(* IEC 61131-3 sources: volt/packages/volt-lsp-iec/test-corpus/bakon-nano/Device/Plc Logic/Application/POUs/MachineControl (part 2) *)

(* ---- MACH_MCL_ModeControl.pou ---- *)
PROGRAM MACH_MCL_ModeControl
VAR
	(* Temporary Variables *)
	bPulseStepCounter	: BOOL;
	bRecipeLoaded		: BOOL;
	tDisableDrives		: TON;
	tonStartButton		: TON;
END_VAR
%LANGUAGE ST
(*************************************************************************
 *
 * Application name				: Snijmachine
 * Module name					: MACH_MCL_ModeControl
 * Version number module		: 0.30
 *
 *
 *						Copyright (c) Bakon 2009
 *						Goes, The Netherlands
 *
 *
 * All rights are reserved. Reproduction in whole or in part is prohibited
 * without the written consent of the copyright owner.
 *
 *************************************************************************)

(*****************************************************************************
 * HISTORY
 *****************************************************************************
 * Update		: 0.20
 * Author		: K.Kole (KOOLE CONTROLS)
 * Changes	: 0.10:	Force to state WaitForInit changed
 *						Condition "bEnableMachine" added in state "WaitForConditioning"
 *				  0.20:	Blockingcounter implemented
 *				  0.30:  Ondelay added for bit g_HMI_bRecipeLoaded in order to avoid
 *						a error in state Wait_For_Automatic
 *****************************************************************************)

	(****************************************************************)
	(*  Mode Control is the central control part of the machines.	*)
	(*  It receives and sends signals from and to the HMI and		 *)
	(*  Handles the signals to and from the machine					  *)
	(****************************************************************)

	(* Hold automatic when ErrorCategory3 *)
	IF			g_sMACH.ERH.bErrorCategory3
	THEN
				g_sMACH.MCL.bHoldOnErrorCat3 := TRUE;
	END_IF
	IF	  	NOT g_sMACH.ERH.bErrorCategory3
		AND	g_HMI_MachCommand.CMD.bStartCycle
	THEN
				 g_sMACH.MCL.bHoldOnErrorCat3 := FALSE;
	END_IF

	(* Stop at end of cycle when ErrorCategory2 *)
	IF				g_sMACH.ERH.bErrorCategory2
	THEN
					g_sMACH.MCL.bStopOnErrorCat2 := TRUE;
	END_IF
	IF	  	NOT	g_sMACH.ERH.bErrorCategory2
		AND NOT	g_sMACH.MCL.bActAutomatic
	THEN
					g_sMACH.MCL.bStopOnErrorCat2 := FALSE;
	END_IF

	(* Stop at end of cycle *)
	IF 	g_HMI_MachCommand.CMD.bStopCycle
	THEN
		g_sMACH.MCL.bStopEndOfCycle := TRUE;
	END_IF
	IF NOT g_sMACH.MCL.bActAutomatic
	THEN
		g_sMACH.MCL.bStopEndOfCycle := FALSE;
	END_IF

	bRecipeLoaded := (g_HMI_sRecipeName <> 'new recipe') AND (g_HMI_sRecipeName <> '');

	(* Recipe downloaded. *)
(*	IF			bRecipeLoaded
		AND (	MACH.MCL.bStateMainSwitchedOn
			OR MACH.MCL.bStateWaitForInit
			OR MACH.MCL.bStateInit
			OR MACH.MCL.bStateWaitForRecipe)
	THEN
		MACH.MCL.bRecipeExecuted := TRUE;
	END_IF
*)
	(* Force StateWaitForAutomatic *)
	IF		  		g_bFirstCycle
		OR NOT 	g_bDI_ES_DirectOK
		OR		g_sMACH.ERR.bTableMovementNotAllowed		// Severe error, chance of damaging the knife
		OR		g_sMACH.ERR.bRAxisMovementNotAllowed		// Severe error, chance of damaging the knife
		OR		g_sMACH.ERR.bZAxisMovementNotAllowed		// Severe error, chance of damaging the knife
		OR		(g_sMACH.ERH.bErrorCategory4
		AND NOT	g_sMACH.MCL.bActManual
		//AND (NOT g_sMACH.MCL.bActAutomatic OR g_bSUB_CleanKnifeStart)
		AND		g_sMACH.MCL.nStepCounter <> StateWaitForAutomatic)
	THEN
				 g_sMACH.MCL.nStepCounter := StateWaitForAutomatic;
	//ELSIF		g_sMACH.ERH.bErrorCategory4			(* Force StateWaitForAuto *)
	//	AND 	g_sMACH.MCL.bActAutomatic
	//	AND NOT	g_bSUB_CleanKnifeStart
	//THEN
	//			 g_sMACH.MCL.nStepCounter := StateWaitForAutomatic;
	END_IF

	(* detect change of state *)
	bPulseStepCounter				:= g_sMACH.MCL.nStepCounter <> g_sMACH.MCL.nOldStepCounter;
	g_sMACH.MCL.nOldStepCounter	:= g_sMACH.MCL.nStepCounter;

IF bPulseStepCounter THEN
	{warning 'Disabled for compatibility SVE'}
	//g_Logger.Write(0, CONCAT('Modecontrol changed to state ', INT_TO_STRING(g_sMACH.MCL.nStepCounter)), 'MACH_MCL_ModeControl');
END_IF

tonStartButton(IN:= g_bDI_StartButton, PT:= T#500MS, Q=> , ET=> );

CASE g_sMACH.MCL.nStepCounter OF
	(* ------------------------------------------------------------------------------
	 * S000 StateMainSwitchedOn
	 *		Reset all Mode Control variables
	 * ------------------------------------------------------------------------------ *)
	StateMainSwitchedOn:

		(* On Entry *)
		IF bPulseStepCounter
		THEN
			g_sMACH.MCL.bActInitialise				:= FALSE;
			g_sMACH.MCL.bActConditioning			:= FALSE;
			g_sMACH.MCL.bActAutomatic			:= FALSE;
			g_sMACH.MCL.bActManual				:= FALSE;
			g_sMACH.MCL.bActCleaning				:= FALSE;
			g_sMACH.MCL.bHoldOnRequest		:= FALSE;
			g_sMACH.MCL.bStopEndOfCycle		:= FALSE;

			(*g_sMACH.MCL.bInitExecuted				:= FALSE; *)
			g_sMACH.MCL.bRecipeExecuted		:= FALSE;
			g_HMI_MachCommand.CMD.bStartManual					:= FALSE;
			g_HMI_MachCommand.CMD.bStartCleaning				:= FALSE;
		  	g_HMI_MachCommand.CMD.bStartCycle				:= FALSE;
		END_IF

		(* Continous actions *)

		(* Transitions *)
		IF				g_bDI_ES_DirectOK
			AND NOT	g_sMACH.ERH.bErrorCategory4
		THEN
			g_sMACH.MCL.nStepCounter := StateWaitForAutomatic;(* StateWaitForInit; *)
			(* On Exit *)
		ELSIF			g_bDI_ES_DirectOK
			AND		g_HMI_MachCommand.CMD.bStartManual
		THEN
			g_sMACH.MCL.nStepCounter := StateManual;
		END_IF

	(* ------------------------------------------------------------------------------
	 * S001 StateWaitForInit
	 *		Wait for init button (No error present )
	 * ------------------------------------------------------------------------------ *)
	StateWaitForInit:

		(* On Entry *)
		IF bPulseStepCounter
		THEN
			(*g_sMACH.MCL.bInitExecuted		:= FALSE; *)
			g_sMACH.MCL.bActInitialise		:= FALSE;
			g_sMACH.MCL.bActConditioning := FALSE;
			g_sMACH.MCL.bActAutomatic	:= FALSE;
			g_sMACH.MCL.bActManual		:= FALSE;
			g_sMACH.MCL.bActCleaning		:= FALSE;
			g_HMI_MachCommand.CMD.bStartManual			:= FALSE;
			g_HMI_MachCommand.CMD.bStartCleaning		:= FALSE;
			g_HMI_MachCommand.CMD.bStartCycle		:= FALSE;

			g_sMACH.MCL.bHoldOnRequest		:= FALSE;
			g_sMACH.MCL.bStopEndOfCycle		:= FALSE;

			tDisableDrives(IN:=FALSE);
			(*g_sMACH.MCL.bRecipeExecuted		:= FALSE; Storing weggelaten dd 1 juni 2011 *)
		END_IF

		(* Continous actions *)
		tDisableDrives(IN:=TRUE, PT:= t#1500ms);
		IF tDisableDrives.Q THEN								(* In AUT, MAN, INI cycles g_uControl_xxx.bAutomatic etc. is reset *)
			g_uControl_X_Axis.bEnableDrive	:= FALSE;			(* Resetting the bEnableDrive bit must be delayed *)
			g_uControl_Y_Axis.bEnableDrive	:= FALSE;
			{warning 'SVE - Check this change}
			//g_uControl_Front_Axis.bEnableDrive	:= g_uStatus_Front_Axis.nStateAxis = 3 OR g_uStatus_Front_Axis.nStateAxis <= 1;			(* Resetting the bEnableDrive bit must be delayed *)
			//g_uControl_Rear_Axis.bEnableDrive	:= g_uStatus_Rear_Axis.nStateAxis = 3 OR g_uStatus_Rear_Axis.nStateAxis <= 1;
			g_uControl_Front_Axis.bEnableDrive := g_uStatus_Front_Axis.eStateAxis <= L_MC1P_AXIS_STATE.StandStill;		//Standstill, Disabled or Errorstop
			g_uControl_Rear_Axis.bEnableDrive := g_uStatus_Rear_Axis.eStateAxis <= L_MC1P_AXIS_STATE.StandStill;		//Standstill, Disabled or Errorstop
			g_uControl_Z_Axis.bEnableDrive	:= FALSE;
			g_uControl_R_Axis.bEnableDrive	:= FALSE;
		END_IF
		(*g_sMACH.ERR.bMoldWarningMold := (NOT FUN_CHECK_MOLD(g_bDI_MoldLeftPresent, g_bDI_MoldRightPresent,(g_HMI_RCP_Parameters.nProductType = Prod_Round),
																			g_bDI_MoldDetection1_1, g_bDI_MoldDetection1_2, g_bDI_MoldDetection1_3,
																			g_bDI_MoldDetection2_1, g_bDI_MoldDetection2_2, g_bDI_MoldDetection2_3,
																			g_HMI_RCP_Parameters.nMaxMoldParts) ) AND (bRecipeLoaded); *)

		(* Transitions *)
		IF 	NOT		g_sMACH.ERH.bError234Active
			AND NOT g_uStatus_X_Axis.bDriveEnabled
			AND NOT g_uStatus_Y_Axis.bDriveEnabled
			AND NOT g_uStatus_Front_Axis.bDriveEnabled
			AND NOT g_uStatus_Rear_Axis.bDriveEnabled
			AND NOT g_uStatus_Z_Axis.bDriveEnabled
			AND NOT g_uStatus_R_Axis.bDriveEnabled
			AND	g_uStatus_R_Axis.bHomePositionAvailable
			AND	(g_HMI_MachCommand.CMD.bStartCycle OR (tonStartButton.Q AND g_HMI_MachCommand.bScanMode))
		THEN
			g_sMACH.MCL.nStepCounter := StateInit;
			(* On Exit *)
		ELSIF g_HMI_MachCommand.CMD.bStartManual						(* Manual *)
		THEN
			g_sMACH.MCL.nStepCounter := StateManual;
		END_IF

	(* ------------------------------------------------------------------------------
	 * S002 StateInit
	 *		Initialising busy
	 * ------------------------------------------------------------------------------ *)
	StateInit:

		(* On Entry *)
		IF bPulseStepCounter
		THEN
			;(*g_sMACH.MCL.bInitExecuted := FALSE; *)
		END_IF

		(* Continous actions *)
		g_sMACH.MCL.bActInitialise := TRUE;

		(* Transitions *)
		IF g_sMACH.uINI.bInitialiseReady
		THEN
			g_sMACH.MCL.nStepCounter := StateWaitForRecipe;
			(* On Exit *)
			g_sMACH.MCL.bActInitialise := FALSE;
			(*g_sMACH.MCL.bInitExecuted  := TRUE; *)
		END_IF

	(* ------------------------------------------------------------------------------
	 * S003 StateWaitForRecipe
	 *		Wait for recipe download
	 * ------------------------------------------------------------------------------ *)
	StateWaitForRecipe:

		(* On Entry *)

		(* Continous actions *)

		(* Transitions *)
		IF bRecipeLoaded						(* Recipe loaded *)
		THEN
			g_sMACH.MCL.nStepCounter := StateWaitForAutomatic;
		ELSIF g_HMI_MachCommand.CMD.bStartManual						(* Manual *)
		THEN
			g_sMACH.MCL.nStepCounter := StateManual;
		ELSIF g_HMI_MachCommand.CMD.bStartCleaning					(* Cleaning *)
		THEN
			g_sMACH.MCL.nStepCounter := StateCleaning;
		END_IF

	(* ------------------------------------------------------------------------------
	 * S004 StateWaitForConditioning
	 *		Wait for start button
	 * ------------------------------------------------------------------------------ *)
(*	StateWaitForConditioning:

		(* On Entry *)
		IF bPulseStepCounter
		THEN
			g_sMACH.MCL.bConditioningExecuted := FALSE;
		END_IF

		(* Continous actions *)

		(* Transitions *)
		IF	g_HMI_MachCommand.CMD.bStartCycle THEN
			g_sMACH.MCL.nStepCounter := StateWaitForAutomatic;
		ELSIF g_HMI_MachCommand.CMD.bStartCycle				  (* Conditioning *)
		THEN
			g_sMACH.MCL.nStepCounter := StateConditioning;
		ELSIF g_sMACH.MCL.bStartInitialise		(* Initialise *)
		THEN
			g_sMACH.MCL.nStepCounter := StateInit;
		ELSIF g_sMACH.MCL.bStartManual			 (* Manual *)
		THEN
			g_sMACH.MCL.nStepCounter := StateManual;
		ELSIF g_sMACH.MCL.bStartCleaning						(* Cleaning *)
		THEN
			g_sMACH.MCL.nStepCounter := StateCleaning;
		END_IF

	(* ------------------------------------------------------------------------------
	 * S005 StateConditioning
	 *		Conditioning busy
	 * ------------------------------------------------------------------------------ *)
	StateConditioning:

		(* On Entry *)
		IF bPulseStepCounter
		THEN
			g_sMACH.MCL.bConditioningExecuted := FALSE;
		END_IF

		(* Continous actions *)
		g_sMACH.MCL.bActConditioning := TRUE;

		(* Transitions *)
		IF (*g_sMACH.CON.BCONDITIONINGREADY*) TRUE
		THEN
			g_sMACH.MCL.nStepCounter := StateWaitForAutomatic;
			(* On Exit *)
			g_sMACH.MCL.bActConditioning		:= FALSE;
			g_sMACH.MCL.bConditioningExecuted := TRUE;
		END_IF
*)
	(* ------------------------------------------------------------------------------
	 * S006 StateWaitForAutomatic
	 *		Wait for start button
	 * ------------------------------------------------------------------------------ *)
	StateWaitForAutomatic:

		(* On Entry *)
		IF bPulseStepCounter
		THEN
			g_sMACH.MCL.bActInitialise		:= FALSE;
			g_sMACH.MCL.bActConditioning := FALSE;
			g_sMACH.MCL.bActAutomatic	:= FALSE;
			g_sMACH.MCL.bActManual		:= FALSE;
			g_sMACH.MCL.bActCleaning		:= FALSE;
			g_HMI_MachCommand.CMD.bStartManual			:= FALSE;
			g_HMI_MachCommand.CMD.bStartCleaning		:= FALSE;
			g_HMI_MachCommand.CMD.bStartCycle		:= FALSE;

			g_sMACH.MCL.bHoldOnRequest		:= FALSE;
			g_sMACH.MCL.bStopEndOfCycle		:= FALSE;

			tDisableDrives(IN:=FALSE);
		END_IF

		(* Continous actions *)
		tDisableDrives(IN:=TRUE, PT:= t#1500ms);
		IF tDisableDrives.Q THEN									(* In AUT, MAN, INI cycles g_uControl_xxx.bAutomatic etc. is reset *)
			g_uControl_X_Axis.bEnableDrive	:= FALSE;			(* Resetting the bEnableDrive bit must be delayed *)
			g_uControl_Y_Axis.bEnableDrive	:= FALSE;
			{warning 'SVE - Check this change}
			//g_uControl_Front_Axis.bEnableDrive	:= g_uStatus_Front_Axis.nStateAxis <> 3 AND g_uStatus_Front_Axis.nStateAxis >= 2;			(* Resetting the bEnableDrive bit must be delayed *)
			//g_uControl_Rear_Axis.bEnableDrive	:= g_uStatus_Rear_Axis.nStateAxis <> 3 AND g_uStatus_Rear_Axis.nStateAxis >= 2;
			g_uControl_Front_Axis.bEnableDrive := g_uStatus_Front_Axis.eStateAxis > L_MC1P_AXIS_STATE.StandStill;	//XX_Motion
			g_uControl_Rear_Axis.bEnableDrive := g_uStatus_Rear_Axis.eStateAxis > L_MC1P_AXIS_STATE.StandStill;	//XX_Motion
			g_uControl_Z_Axis.bEnableDrive	:= FALSE;
			g_uControl_R_Axis.bEnableDrive	:= FALSE;
		END_IF;

		(* Transitions *)
		IF				(g_HMI_MachCommand.CMD.bStartCycle  OR (tonStartButton.Q AND g_HMI_MachCommand.bScanMode))					(* Start auto cycle *)
			AND NOT	g_sMACH.MCL.bStopOnErrorCat2
			AND NOT	g_sMACH.MCL.bHoldOnErrorCat3
			AND		g_bAxis_FrontSet								(* Axis referenced to zero (in manual page) *)
			AND		g_bAxis_RearSet								(* Axis referenced to zero (in manual page) *)
			AND		g_bAxis_RSet									(* Axis referenced to zero (in manual page) *)
			AND		((g_sHMI_CountersInfinite.dnHourCount <= g_HMI_MCH_dnBlockCounter) OR (g_HMI_MCH_dnBlockCounter = 0))
		THEN
			g_sMACH.MCL.nStepCounter := StateAutomatic;
		ELSIF g_HMI_MachCommand.CMD.bStartManual								(* Manual *)
		THEN
			g_sMACH.MCL.nStepCounter := StateManual;
		ELSIF g_HMI_MachCommand.CMD.bStartCleaning							(* Cleaning *)
		THEN
			g_sMACH.MCL.nStepCounter := StateCleaning;
		END_IF

	(* ------------------------------------------------------------------------------
	 * S007 StateAutomatic
	 *		Automatic busy
	 * ------------------------------------------------------------------------------ *)
	StateAutomatic:

		(* On Entry *)

		(* Continous actions *)
		g_sMACH.MCL.bActAutomatic := TRUE;
		IF	g_HMI_MachCommand.CMD.bPauseCycle
		THEN
			g_sMACH.MCL.bHoldOnRequest := TRUE;
		END_IF
		IF	g_HMI_MachCommand.CMD.bStartCycle
		THEN
			g_sMACH.MCL.bHoldOnRequest := FALSE;
		END_IF

		(* Transitions *)
		IF g_sMACH.AUT.bAutomaticReady
		THEN
			g_sMACH.MCL.nStepCounter := StateWaitForAutomatic;
			(* On Exit *)
			g_sMACH.MCL.bActAutomatic			:= FALSE;
			g_sMACH.MCL.bHoldOnRequest		:= FALSE;
		END_IF

	(* ------------------------------------------------------------------------------
	 * S008 StateManual
	 *		Manual mode busy
	 * ------------------------------------------------------------------------------ *)
	StateManual:

		(* On Entry *)
		IF bPulseStepCounter
		THEN
			g_sMACH.MCL.bActManual := TRUE;
		END_IF

		(* Continous actions *)
		g_HMI_MachCommand.CMD.bStartManual	:= FALSE;
		IF 	g_HMI_MachCommand.CMD.bStopManual
		THEN
			g_sMACH.MCL.bStopEndOfCycle := TRUE;
		END_IF

		(* Transitions *)
		IF g_sMACH.MAN.bManualReady
		THEN
			g_sMACH.MCL.bActManual := FALSE;
			g_sMACH.MCL.nStepCounter := StateWaitForAutomatic;	(* StateWaitForInit; *)
		END_IF

	(* ------------------------------------------------------------------------------
	 * S009 StateCleaning
	 *		Cleaning mode busy
	 * ------------------------------------------------------------------------------ *)
	StateCleaning:

		(* On Entry *)
		IF bPulseStepCounter
		THEN
			g_sMACH.MCL.bActCleaning := TRUE;
			g_HMI_MachCommand.CMD.bStopCleaning	:= FALSE;
		END_IF

		(* Continous actions *)
		IF	g_HMI_MachCommand.CMD.bStopCleaning
		THEN
			g_sMACH.MCL.bStopEndOfCycle := TRUE;
		END_IF

		(* Transitions *)
		IF	g_sMACH.CLN.bCleaningReady
		THEN
			g_sMACH.MCL.bActCleaning := FALSE;
			g_HMI_MachCommand.CMD.bStopCleaning	:= FALSE;
			g_sMACH.MCL.nStepCounter := StateWaitForAutomatic;	(*StateWaitForInit; *)
		END_IF

	END_CASE

END_PROGRAM

(* ---- MACH_MIS_Miscellaneous.pou ---- *)
PROGRAM MACH_MIS_Miscellaneous
VAR
	TONMinute: TON;
	bMinute	: BOOL;

END_VAR
%LANGUAGE ST
(* Machine producing hours *)
TONMinute(IN:=g_sMACH.AUT.bActAutomatic AND NOT bMinute, PT:=T#60s);
bMinute := TONMinute.Q;
IF bMinute THEN
	 g_sHMI_CountersInfinite.nMinuteCount := g_sHMI_CountersInfinite.nMinuteCount + 1;
END_IF
IF g_sHMI_CountersInfinite.nMinuteCount >= 60 THEN
	g_sHMI_CountersInfinite.nMinuteCount := 0;
	g_sHMI_CountersInfinite.dnHourCount := g_sHMI_CountersInfinite.dnHourCount + 1;
END_IF

(* Maintenance necessary after x running hours *)
g_sMACH.ERR.bMaintenanceNecessary := 			g_sHMI_CountersInfinite.dnHourCount >= (g_HMI_dnLastMaintenance + g_HMI_MCH_Parameters.dnMaintenanceInterval)
											AND	g_HMI_MCH_Parameters.dnMaintenanceInterval > 0;
IF g_HMI_MachCommand.CMD.bMaintenanceDone
THEN
	g_HMI_dnLastMaintenance := g_sHMI_CountersInfinite.dnHourCount;
END_IF

IF			g_HMI_nDefaultLanguage <> 1043	(* nederlands *)
	AND	g_HMI_nDefaultLanguage <> 1033	(* engels *)
	AND	g_HMI_nDefaultLanguage <> 1031	(* duits *)
	AND	g_HMI_nDefaultLanguage <> 1034	(* spaans *)
	AND	g_HMI_nDefaultLanguage <> 1036	(* frans *)
	AND g_HMI_nDefaultLanguage <> 1040	(* Italiaans*)
	AND	g_HMI_nDefaultLanguage <> 1045	(* pools *)
	AND	g_HMI_nDefaultLanguage <> 1048	(* roemeens *)
	AND g_HMI_nDefaultLanguage <> 1049	(* Russian*)
	AND	g_HMI_nDefaultLanguage <> 1050	(* kroatisch *)
	AND g_HMI_nDefaultLanguage <> 1061	(* Ests*)
	AND g_HMI_nDefaultLanguage <> 2052	(* Chinees*)
	AND g_HMI_nDefaultLanguage <> 1029	(* Tsjechisch*)
	AND g_HMI_nDefaultLanguage <> 2070	(* Portugees*)
	AND g_HMI_nDefaultLanguage <> 1053	(* Zweeds *)

THEN
	g_sMACH.ERR.bLanguageValueInvalid	:= TRUE;
END_IF
IF	g_sMACH.ERR.bLanguageValueInvalid
THEN
	g_HMI_nDefaultLanguage := 1033;	(* English, US *)
END_IF

END_PROGRAM

(* ---- MACH_SUB_CleanCycle.pou ---- *)
PROGRAM MACH_SUB_CleanCycle
VAR
	bPulseStepCounter		: BOOL;
	bWait					: BOOL;
	bTableToSafeCleanPos	: BOOL;
	bCleanWithScraper		: BOOL;
	bCleanWithWater			: BOOL;
	rSafePosX				: REAL;
	tWatchDogTimer			: TON;
	tStepTimer				: TOF;
END_VAR

%LANGUAGE ST
(*************************************************************************
 *
 * Application name				: Snijmachine Quintens
 * Module name					: MACH_Sub_CleanCycle
 * Version number module		: 0.10
 *
 *
 *						Copyright (c) Bakon 2009
 *						Goes, The Netherlands
 *
 *
 * All rights are reserved. Reproduction in whole or in part is prohibited
 * without the written consent of the copyright owner.
 *
 *************************************************************************)

(*************************************************************************
 * HISTORY
 *************************************************************************
 * Update 	: 0.10
 * Author 	: K. Kole
 *************************************************************************)

(* Force C_NOT_ACTIVE state *)
IF	  NOT 	g_bSUB_CleanKnifeStart
THEN
			g_sMACH.SUBClean.nStepCounter := C_NOT_ACTIVE;
END_IF;

IF			g_sMACH.SUBClean.nStepCounter <> C_NOT_ACTIVE
THEN
	(* -------------------------------------------------------------------------
	 * Prestep Code
	 * ------------------------------------------------------------------------- *)
				  ;
END_IF;

(* detect change of state *)
bPulseStepCounter			  := g_sMACH.SUBClean.nStepCounter <> g_sMACH.SUBClean.nOldStepCounter;
g_sMACH.SUBClean.nOldStepCounter := g_sMACH.SUBClean.nStepCounter;

(* Steptimer *)
tStepTimer (IN:= bPulseStepCounter, PT:= REAL_TO_TIME(g_sMACH.SUBClean.rStepTime));
bWait := tStepTimer.Q;

(* Watchdogtimer *)
tWatchDogTimer (IN:= 	NOT	bPulseStepCounter
						AND		g_bSUB_CleanKnifeStart
						AND NOT	g_HMI_MachCommand.CMD.bResetErrorPulse
						AND		g_sMACH.SUBClean.rWatchdogTime <> 0,
					PT:= REAL_TO_TIME(g_sMACH.SUBClean.rWatchdogTime));
g_sMACH.SUBClean.bAlmError := tWatchDogTimer.Q;

g_sMACH.SUBClean.bSubProcessBusy1	:= bTableToSafeCleanPos;
rSafePosX	:= 2.1;

CASE g_sMACH.SUBClean.nStepCounter OF
	(* --------------------------------------------------------------------------
	 * S-1  C_NOT_ACTIVE
	 *		OnEntry: Ready  := FALSE
	 *		OnEntry: Busy	:= FALSE
	 *		OnEntry: Reset all non-stored commands
	 * T000 Activate signal
	 * -------------------------------------------------------------------------- *)
	C_NOT_ACTIVE:

		(* On Entry *)
		IF		bPulseStepCounter
		THEN
				g_sMACH.SUBClean.rWatchdogTime	:= 0;
				g_sMACH.SUBClean.bSubReady		:= FALSE;
				g_sMACH.SUBClean.bSubBusy		:= FALSE;

				g_bSUB_CleanKnifeDone			:= FALSE;

				g_sMACH.SUBClean.bPreventAction	:= FALSE;

				//g_uControl_X_Axis.bEnableDrive				:= FALSE;
				g_uControl_X_Axis.bPosABSPosition			:= FALSE;

				//g_uControl_Y_Axis.bEnableDrive				:= FALSE;
				g_uControl_Y_Axis.bPosABSPosition			:= FALSE;

				//g_uControl_Z_Axis.bEnableDrive				:= FALSE;
				g_uControl_Z_Axis.bStartHoming				:= FALSE;
				g_uControl_Z_Axis.bPosABSPosition			:= FALSE;	(* Used only after axis has first been homed to its sensor *)

				//g_uControl_R_Axis.bEnableDrive				:= FALSE;
				g_uControl_R_Axis.bPosABSPosition			:= FALSE;

				g_sMACH.sCleaningContainerControl.bPosExecute := FALSE;
				g_bDQ_CleaningWaterValve					:= FALSE;
				g_bDQ_CleaningAirValve := FALSE;
				//g_bCMD_US_Start1 							:= FALSE;
				g_bUS_EnableCleaning						:= FALSE;

				bTableToSafeCleanPos						:= FALSE;		(* Move table to safe position only, thus no cleaning of knife *)
		END_IF

		(* Continuous actions *)
		bCleanWithScraper	:=		(g_HMI_RCP_Parameters.nCleanWithScraper <= 1)		// Recipe value only valid at beginning of cycle
								OR	g_sMACH.MCL.bActCleaning;							// In cleaning mode scraper always in use
		bCleanWithWater		:=		(g_HMI_RCP_Parameters.nCleanWithScraper <> 1)
								OR  g_sMACH.MCL.bActCleaning;

		(* Transitions *)
		IF		g_bSUB_CleanKnifeStart
		THEN
				g_uControl_X_Axis.bEnableDrive		:= TRUE;
				g_uControl_Y_Axis.bEnableDrive		:= TRUE;
				g_uControl_Front_Axis.bEnableDrive	:= TRUE;
				g_uControl_Rear_Axis.bEnableDrive	:= TRUE;
				g_uControl_Z_Axis.bEnableDrive		:= TRUE;
				g_uControl_R_Axis.bEnableDrive		:= TRUE;
				IF		g_sMACH.MCL.bActCleaning
					AND	g_HMI_MachCommand.CMD.bTableToCleanPos
				THEN
					bTableToSafeCleanPos	:= TRUE;		(* Move table to safe position only, thus no cleaning of knife *)
				END_IF
				g_sMACH.SUBClean.nStepCounter		:= C_INITIAL;
		END_IF

	(* --------------------------------------------------------------------------
	 * S000 C_INITIAL
	 *		OnEntry: Ready := FALSE
	 *		OnEntry: Busy  := TRUE
	 * T001 Always
	 * -------------------------------------------------------------------------- *)
	C_INITIAL:

		(* On Entry *)
		IF			bPulseStepCounter
		THEN
					g_sMACH.SUBClean.rWatchdogTime		:= 10 * 1000;
					g_sMACH.SUBClean.bSubReady			:= FALSE;
					g_sMACH.SUBClean.bSubBusy			:= TRUE;
		END_IF

		(* Continuous actions *)
		IF g_sMACH.SUBClean.bAlmError THEN
			IF NOT g_uStatus_X_Axis.bDriveEnabled
				OR NOT g_uStatus_Y_Axis.bDriveEnabled
				OR NOT g_uStatus_Front_Axis.bDriveEnabled
				OR NOT g_uStatus_Rear_Axis.bDriveEnabled
			THEN
				g_sMACH.ERR.bXYNotEnabled := TRUE;
			END_IF
			IF NOT g_uStatus_Z_Axis.bDriveEnabled THEN
				g_sMACH.ERR.bZNotEnabled := TRUE;
			END_IF
			IF NOT g_uStatus_R_Axis.bDriveEnabled THEN
				g_sMACH.ERR.bRNotEnabled := TRUE;
			END_IF
		END_IF

		(* Transitions *)
		IF		g_uStatus_Z_Axis.bDriveEnabled// AND g_uStatus_Z_Axis.bAutomaticEnabled
			AND	g_uStatus_R_Axis.bDriveEnabled //AND g_uStatus_R_Axis.bAutomaticEnabled
			AND	g_uStatus_X_Axis.bDriveEnabled //AND g_uStatus_X_Axis.bAutomaticEnabled
			AND	g_uStatus_Y_Axis.bDriveEnabled //AND g_uStatus_Y_Axis.bAutomaticEnabled
			AND	g_uStatus_Rear_Axis.bDriveEnabled //AND g_uStatus_Rear_Axis.bAutomaticEnabled
			AND	g_uStatus_Front_Axis.bDriveEnabled //AND g_uStatus_Front_Axis.bAutomaticEnabled
		THEN
			g_sMACH.SUBClean.nStepCounter	:= 005;
		END_IF

	(* --------------------------------------------------------------------------
	 * S005 Move Z to safe position
	 * T010 Z axis busy
	 * -------------------------------------------------------------------------- *)
	005:

		(* On Entry *)
		IF		 bPulseStepCounter
		THEN
				g_sMACH.SUBClean.rWatchdogTime		:= 0;
				g_sMACH.SUBClean.rStepTime			:= 0;
				g_uControl_Z_Axis.lrPosition		:= g_sCalculated.rAboveProductPos;
				g_uControl_Z_Axis.bPosABSPosition	:= TRUE;
		END_IF

		(* Continuous actions *)

		(* Transitions *)
		IF		g_uStatus_Z_Axis.bMoveAbsDone
		THEN
				g_sMACH.SUBClean.nStepCounter				:= 010;
		END_IF

	(* --------------------------------------------------------------------------
	 * S010 Wait Z positioning to safe pos done
	 * T015 Z axis positioning done
	 * -------------------------------------------------------------------------- *)
	010:

		(* On Entry *)
		IF		 bPulseStepCounter
		THEN
				g_sMACH.SUBClean.rWatchdogTime		:= 0;
				g_sMACH.SUBClean.rStepTime			:= 0;
		END_IF

		(* Continuous actions *)

		(* Transitions *)
		IF			g_uStatus_Z_Axis.bMoveAbsDone
		THEN
					g_uControl_Z_Axis.bPosABSPosition	:= FALSE;
					g_sMACH.SUBClean.nStepCounter		:= 015;
		END_IF

	(* --------------------------------------------------------------------------
	 * S015 Move cleaning cylinder down.
	 * T020 Cleaning cylinder busy
	 * -------------------------------------------------------------------------- *)
	015:

		(* On Entry *)
		IF		 bPulseStepCounter
		THEN
				g_sMACH.SUBClean.rWatchdogTime		:= 0;
				g_sMACH.SUBClean.rStepTime			:= 100;
				g_sMACH.sCleaningContainerControl.rTargetPosition := 0;
				g_sMACH.sCleaningContainerControl.bPosExecute := gMachConfig.bCleaningUnit;
		END_IF

		(* Continuous actions *)

		(* Transitions *)
		IF	NOT bWait
		THEN
					g_sMACH.SUBClean.nStepCounter		:= 020;
		END_IF

	(* --------------------------------------------------------------------------
	 * S020 Wait for R positioning to 90 dgrees done
	 * T025 R-axis positioning done AND NOT bTableToCleanPos
	 * T040 R-axis positioning done AND bTableToCleanPos
	 * -------------------------------------------------------------------------- *)
	020:

		(* On Entry *)
		IF		 bPulseStepCounter
		THEN
				g_sMACH.SUBClean.rWatchdogTime		:= 0;
				g_sMACH.SUBClean.rStepTime			:= 0;
		END_IF

		(* Continuous actions *)

		(* Transitions *)
		IF	(g_sMACH.sCleaningContainerStatus.rActualPosition = 0 OR NOT gMachConfig.bCleaningUnit)
		THEN
				g_sMACH.sCleaningContainerControl.bPosExecute	:= FALSE;
				g_sMACH.SUBClean.nStepCounter			:= 025;
		END_IF

	(* --------------------------------------------------------------------------
	 * S025 Move X to start position or to Safe pos X (2.1)
	 *		Move Y to start cleaning position OR End cleaning position when TableToSafePos or Not UseScraper
	 *		Move R to 90 degrees and cleaning cylinder down.
	 * T030 X, Y and R axis ready
	 * -------------------------------------------------------------------------- *)
	025:

		(* On Entry *)
		IF		 bPulseStepCounter
		THEN
				g_sMACH.SUBClean.rWatchdogTime		:= 0;
				g_sMACH.SUBClean.rStepTime			:= 0;
				IF	bTableToSafeCleanPos THEN
					g_uControl_X_Axis.lrPosition		:= rSafePosX;
					g_uControl_Y_Axis.lrPosition		:= g_HMI_MCH_Parameters.rCleanYPosStop;
				ELSIF NOT bCleanWithScraper THEN
					g_uControl_X_Axis.lrPosition		:= rSafePosX;
					g_uControl_Y_Axis.lrPosition		:= g_HMI_MCH_Parameters.rCleanYPosStop;
				ELSE
					g_uControl_X_Axis.lrPosition		:= g_HMI_MCH_Parameters.rCleanXPosStart;
					g_uControl_Y_Axis.lrPosition		:= g_HMI_MCH_Parameters.rCleanYPosStart;
				END_IF
				g_uControl_X_Axis.bPosABSPosition	:= TRUE;
				g_uControl_Y_Axis.bPosABSPosition	:= TRUE;
				g_uControl_R_Axis.lrPosition		:= 90;
				g_uControl_R_Axis.bPosABSPosition	:= TRUE;
		END_IF

		(* Continuous actions *)

		(* Transitions *)
		IF			g_uStatus_R_Axis.bMoveAbsDone
			AND		g_uStatus_Y_Axis.bMoveAbsDone
			AND		g_uStatus_X_Axis.bMoveAbsDone
			AND		(g_uStatus_X_Axis.lrActPosition < g_HMI_MCH_Parameters.rCleanXPosStart + 1)		// "Dubbele" controle...
		THEN
					g_uControl_X_Axis.bPosABSPosition	:= FALSE;
					g_uControl_Y_Axis.bPosABSPosition	:= FALSE;
					g_uControl_R_Axis.bPosABSPosition	:= FALSE;
					IF	bTableToSafeCleanPos THEN
						g_sMACH.SUBClean.nStepCounter		:= C_READY;
					ELSIF NOT bCleanWithScraper THEN
						g_sMACH.SUBClean.nStepCounter		:= 045;
					ELSE
						g_sMACH.SUBClean.nStepCounter		:= 030;
					END_IF
		END_IF

	(* --------------------------------------------------------------------------
	 * S030 Move Z t cleaning position
	 * T035 Z axis ready and clean with scraper
	 * T040 Z axis ready and clean without scraper
	 * -------------------------------------------------------------------------- *)
	030:

		(* On Entry *)
		IF		 bPulseStepCounter
		THEN
				g_sMACH.SUBClean.rWatchdogTime		:= 0;
				g_sMACH.SUBClean.rStepTime			:= 0;
				g_uControl_Z_Axis.lrPosition		:= g_HMI_MCH_Parameters.rCleanZPosFlap;
				g_uControl_Z_Axis.bPosABSPosition	:= TRUE;
		END_IF

		(* Continuous actions *)

		(* Transitions *)
		IF			g_uStatus_Z_Axis.bMoveAbsDone
		THEN
					g_uControl_Z_Axis.bPosABSPosition	:= FALSE;
					g_sMACH.SUBClean.nStepCounter		:= 035;
		END_IF

	(* --------------------------------------------------------------------------
	 * S035 Start positioning Y to end position
	 * T040 Y axis ready
	 * -------------------------------------------------------------------------- *)
	035:

		(* On Entry *)
		IF		 bPulseStepCounter
		THEN
				g_sMACH.SUBClean.rWatchdogTime		:= 0;
				g_sMACH.SUBClean.rStepTime			:= 0;
				g_uControl_Y_Axis.lrPosition		:= g_HMI_MCH_Parameters.rCleanYPosStop;
				g_uControl_Y_Axis.bPosABSPosition	:= TRUE;
		END_IF

		(* Continuous actions *)

		(* Transitions *)
		IF			g_uStatus_Y_Axis.bMoveAbsDone
		THEN
					g_uControl_Y_Axis.bPosABSPosition	:= FALSE;
					g_sMACH.SUBClean.nStepCounter		:= 040;
		END_IF

	(* --------------------------------------------------------------------------
	 * S040 Start positioning X to safe position
	 * T045 X axis ready
	 * -------------------------------------------------------------------------- *)
	040:

		(* On Entry *)
		IF		 bPulseStepCounter
		THEN
				g_sMACH.SUBClean.rWatchdogTime		:= 0;
				g_sMACH.SUBClean.rStepTime			:= 0;
				g_uControl_X_Axis.lrPosition		:= rSafePosX;		(* Fixed position!! *)
				g_uControl_X_Axis.bPosABSPosition	:= TRUE;
		END_IF

		(* Continuous actions *)

		(* Transitions *)
		IF		g_uStatus_X_Axis.bMoveAbsDone
		THEN
				g_uControl_X_Axis.bPosABSPosition	:= FALSE;
				IF bCleanWithWater THEN
					g_sMACH.SUBClean.nStepCounter		:= 45;
				ELSE
					g_sMACH.SUBClean.nStepCounter		:= 065;
				END_IF
		END_IF

	(* --------------------------------------------------------------------------
	 * S045 Move Cleaning unit up and move Z-axis to spray water position
	 * T050 Cleaning unit up
	 * -------------------------------------------------------------------------- *)
	045:

		(* On Entry *)
		IF		 bPulseStepCounter
		THEN
				g_sMACH.SUBClean.rWatchdogTime		:= 0;
				g_sMACH.SUBClean.rStepTime			:= 0;
				g_sMACH.sCleaningContainerControl.rTargetPosition := 1;
				g_sMACH.sCleaningContainerControl.bPosExecute := gMachConfig.bCleaningUnit;
				g_uControl_Z_Axis.lrPosition		:= g_HMI_MCH_Parameters.rCleanZPosWaterContainer;
				g_uControl_Z_Axis.bPosABSPosition	:= TRUE;
		END_IF

		(* Continuous actions *)

		(* Transitions *)
		IF			g_sMACH.sCleaningContainerStatus.rActualPosition = 1
				AND	g_uStatus_Z_Axis.bMoveAbsDone
		THEN
					g_uControl_Z_Axis.bPosABSPosition	:= FALSE;
					g_sMACH.sCleaningContainerControl.bPosExecute	:= FALSE;
					g_sMACH.SUBClean.nStepCounter		:= 050;
		END_IF

	(* --------------------------------------------------------------------------
	 * S050 Start spraying water
	 * T055 Water spraying ready
	 * -------------------------------------------------------------------------- *)
	050:

		(* On Entry *)
		IF		 bPulseStepCounter
		THEN
				g_sMACH.SUBClean.rWatchdogTime		:= 0;
				g_sMACH.SUBClean.rStepTime			:= g_HMI_RCP_Parameters.rCleaningTimeWater * 1000;
				g_bDQ_CleaningWaterValve			:= TRUE;
		END_IF

		(* Continuous actions *)

		(* Transitions *)
		IF		NOT bWait
		THEN
				g_bDQ_CleaningWaterValve			:= FALSE;
				g_sMACH.SUBClean.nStepCounter		:= 052;
		END_IF

	(* --------------------------------------------------------------------------
	 * S052 Activate ultrasonic
	 * T053 Ultrasonic ready
	 * -------------------------------------------------------------------------- *)
	052:

		(* On Entry *)
		IF		 bPulseStepCounter
		THEN
				g_sMACH.SUBClean.rWatchdogTime		:= 0;
				g_sMACH.SUBClean.rStepTime			:= g_HMI_RCP_Parameters.rCleaningTimeUltrasonic * 1000;
				//g_bCMD_US_Start1 					:= TRUE;
				g_bUS_EnableCleaning				:= TRUE;
		END_IF

		(* Continuous actions *)

		(* Transitions *)
		IF		NOT bWait
		THEN
				//g_bCMD_US_Start1 					:= FALSE;
				g_bUS_EnableCleaning				:= FALSE;
				g_sMACH.SUBClean.nStepCounter		:= 053;
		END_IF

	(* --------------------------------------------------------------------------
	 * S053 Start spraying air
	 * T055 Air spraying done
	 * -------------------------------------------------------------------------- *)
	053:

		(* On Entry *)
		IF		 bPulseStepCounter
		THEN
				g_sMACH.SUBClean.rWatchdogTime		:= 0;
				g_sMACH.SUBClean.rStepTime			:= g_HMI_RCP_Parameters.rCleaningTimeAir * 1000;
				g_bDQ_CleaningAirValve			:= TRUE;
		END_IF

		(* Continuous actions *)

		(* Transitions *)
		IF		NOT bWait
		THEN
				g_sMACH.SUBClean.nStepCounter		:= 055;
		END_IF

	(* --------------------------------------------------------------------------
	 * S055 Move Cleaning unit down (safe position)
	 * T060 X axis ready
	 * -------------------------------------------------------------------------- *)
	055:

		(* On Entry *)
		IF		 bPulseStepCounter
		THEN
				g_sMACH.SUBClean.rWatchdogTime		:= 0;
				g_sMACH.SUBClean.rStepTime			:= 0;
				g_sMACH.sCleaningContainerControl.rTargetPosition := 0;
				g_sMACH.sCleaningContainerControl.bPosExecute := gMachConfig.bCleaningUnit;
		END_IF

		(* Continuous actions *)

		(* Transitions *)
		IF			g_sMACH.sCleaningContainerStatus.rActualPosition = 0 OR NOT gMachConfig.bCleaningUnit
		THEN
					g_bDQ_CleaningAirValve := FALSE;
					g_sMACH.sCleaningContainerControl.bPosExecute	:= FALSE;
					g_sMACH.SUBClean.nStepCounter		:= 065;
		END_IF

	(* --------------------------------------------------------------------------
	 * S065 Move Z to safe position
	 * READY Z axis done and automatic
	 * -------------------------------------------------------------------------- *)
	065:

		(* On Entry *)
		IF		 bPulseStepCounter
		THEN
				g_sMACH.SUBClean.rWatchdogTime			:= 0;
				g_sMACH.SUBClean.rStepTime				:= 0;
				g_uControl_Z_Axis.lrPosition			:= g_sCalculated.rAboveProductPos;
				g_uControl_Z_Axis.bPosABSPosition	:= TRUE;
		END_IF

		(* Continuous actions *)

		(* Transitions *)
		IF		g_uStatus_Z_Axis.bMoveAbsDone
		THEN
				g_uControl_Z_Axis.bPosABSPosition	:= FALSE;
				IF g_sMACH.MCL.bActAutomatic THEN
					g_sMACH.SUBClean.nStepCounter		:= C_READY;
				ELSE
					g_sMACH.SUBClean.nStepCounter		:= 070;
				END_IF
		END_IF

	(* --------------------------------------------------------------------------
	 * S070 Start positioning Y to pre infeed position (+ 30)
	 * T075 Y axis ready
	 * -------------------------------------------------------------------------- *)
	070:

		(* On Entry *)
		IF		 bPulseStepCounter
		THEN
				g_sMACH.SUBClean.rWatchdogTime		:= 0;
				g_sMACH.SUBClean.rStepTime			:= 0;
				g_uControl_Y_Axis.lrPosition		:= g_HMI_MCH_Parameters.rInfeedPosition_Y + 30;
				g_uControl_Y_Axis.bPosABSPosition	:= TRUE;
		END_IF

		(* Continuous actions *)

		(* Transitions *)
		IF			g_uStatus_Y_Axis.bMoveAbsDone
		THEN
					g_uControl_Y_Axis.bPosABSPosition	:= FALSE;
					g_sMACH.SUBClean.nStepCounter		:= 075;
		END_IF

	(* --------------------------------------------------------------------------
	 * S075 Start homing X, R to zero
	 * T080 X axis ready
	 * -------------------------------------------------------------------------- *)
	075:

		(* On Entry *)
		IF		 bPulseStepCounter
		THEN
				g_sMACH.SUBClean.rWatchdogTime		:= 0;
				g_sMACH.SUBClean.rStepTime			:= 0;
				g_uControl_X_Axis.lrPosition		:= g_HMI_MCH_Parameters.rInfeedPosition_X;
				g_uControl_X_Axis.bPosABSPosition	:= TRUE;
				g_uControl_R_Axis.lrPosition		:= 0;
				g_uControl_R_Axis.bPosABSPosition	:= TRUE;
		END_IF

		(* Continuous actions *)

		(* Transitions *)
		IF			g_uStatus_X_Axis.bMoveAbsDone
			AND		g_uStatus_R_Axis.bMoveAbsDone
		THEN
					g_uControl_X_Axis.bPosABSPosition	:= FALSE;
					g_uControl_R_Axis.bPosABSPosition	:= FALSE;
					//IF g_sMACH.MCL.bActAutomatic THEN
					//	g_sMACH.SUBClean.nStepCounter		:= 80;
					//ELSE
						g_sMACH.SUBClean.nStepCounter		:= C_READY;
					//END_IF
		END_IF

	(* --------------------------------------------------------------------------
	 * S080 Start homing Y
	 * Ready Y axis ready
	 * -------------------------------------------------------------------------- *)
	080:

		(* On Entry *)
		IF		 bPulseStepCounter
		THEN
				g_sMACH.SUBClean.rWatchdogTime		:= 0;
				g_sMACH.SUBClean.rStepTime			:= 0;
				g_uControl_Y_Axis.lrPosition		:= g_HMI_MCH_Parameters.rInfeedPosition_Y;
				g_uControl_Y_Axis.bPosABSPosition	:= TRUE;
		END_IF

		(* Continuous actions *)

		(* Transitions *)
		IF		g_uStatus_Y_Axis.bMoveAbsDone
		THEN
				g_uControl_Y_Axis.bPosABSPosition	:= FALSE;
				g_sMACH.SUBClean.nStepCounter		:= C_READY;
		END_IF

	(* --------------------------------------------------------------------------
	 * S998 C_READY
	 *		OnEntry: Ready		:= TRUE
	 *		OnEntry: Busy		 := FALSE
	 *		Always : Activate errorhandler
	 * T000 Never
	 * -------------------------------------------------------------------------- *)
	C_READY:

		(* On Entry *)
		IF		bPulseStepCounter
		THEN
				g_sMACH.SUBClean.rWatchdogTime	:= 0;
				g_sMACH.SUBClean.bSubReady		:= TRUE;
				g_sMACH.SUBClean.bSubBusy		:= FALSE;
		END_IF

		(* Continuous actions *)
		g_bSUB_CleanKnifeDone							:= TRUE;

		(* Transitions *)
		IF			FALSE
		THEN
					g_sMACH.SUBClean.nStepCounter		:= C_INITIAL;
		END_IF

(* --------------------------------------------------------------------------
 * Illegal state
 * -------------------------------------------------------------------------- *)
ELSE
	(* Programming error: Illegal state *)
	g_sMACH.SUBClean.rWatchdogTime := 10;
END_CASE;

IF			g_sMACH.SUBClean.nStepCounter <> C_NOT_ACTIVE
THEN
	(* -------------------------------------------------------------------------
	 * Poststep Code
	 * ------------------------------------------------------------------------- *)
	;
END_IF

END_PROGRAM

(* ---- MACH_SUB_Initialise.pou ---- *)
PROGRAM MACH_SUB_Initialise
VAR
	bPulseStepCounter		: BOOL;
	bWait					: BOOL;
	tWatchDogTimer			: TON;
	tStepTimer				: TOF;
	tDelayStep5				: TON;
END_VAR
VAR_INPUT
	I_rX_InfeedPosition		: REAL;
	I_rY_InfeedPosition		: REAL;
	I_rY_InfeedPrePosition	: REAL;
END_VAR
%LANGUAGE ST
(*************************************************************************
 *
 * Application name				: Snijmachine
 * Module name					: MACH_SUB_Initialise
 * Version number module		: 0.00
 *
 *
 *						Copyright (c) Bakon 2009
 *						Goes, The Netherlands
 *
 *
 * All rights are reserved. Reproduction in whole or in part is prohibited
 * without the written consent of the copyright owner.
 *
 *************************************************************************)

(*************************************************************************
 * HISTORY
 *************************************************************************
 * Update  : 0.00
 * Author  :	 K. Kole
 * Changes :
 *************************************************************************)

(* Force C_NOT_ACTIVE state *)
IF	  NOT g_bSUB_InitStart
THEN
		  g_sMACH.SUBInit.nStepCounter := C_NOT_ACTIVE;
END_IF

IF		g_sMACH.SUBInit.nStepCounter <> C_NOT_ACTIVE
THEN
	(* -------------------------------------------------------------------------
	 * Prestep Code
	 * ------------------------------------------------------------------------- *)
				  ;
END_IF

(* detect change of state *)
bPulseStepCounter	  := g_sMACH.SUBInit.nStepCounter <> g_sMACH.SUBInit.nOldStepCounter;
g_sMACH.SUBInit.nOldStepCounter := g_sMACH.SUBInit.nStepCounter;

(* Steptimer *)
tStepTimer (IN:= bPulseStepCounter, PT:= REAL_TO_TIME(g_sMACH.SUBInit.rStepTime));
bWait := tStepTimer.Q;

(* Watchdogtimer *)
tWatchDogTimer (IN:= 	NOT	bPulseStepCounter
						AND		g_bSUB_InitStart
						AND NOT	g_HMI_MachCommand.CMD.bResetErrorPulse
						AND		g_sMACH.SUBInit.rWatchdogTime <> 0,
					PT:= REAL_TO_TIME(g_sMACH.SUBInit.rWatchdogTime));
g_sMACH.SUBInit.bAlmError := tWatchDogTimer.Q;

tDelayStep5(IN:= , PT:= T#200MS, Q=> , ET=> );

CASE g_sMACH.SUBInit.nStepCounter OF
	(* --------------------------------------------------------------------------
	 * S-1  C_NOT_ACTIVE
	 *		OnEntry: Ready  := FALSE
	 *		OnEntry: Busy	:= FALSE
	 *		OnEntry: Reset all non-stored commands
	 * T000 Activate signal
	 * -------------------------------------------------------------------------- *)
	C_NOT_ACTIVE:

		(* On Entry *)
		IF		bPulseStepCounter
		THEN
				g_sMACH.SUBInit.rWatchdogTime				:= 0;
				g_sMACH.SUBInit.bSubReady					:= FALSE;
				g_sMACH.SUBInit.bSubBusy					:= FALSE;

				g_bSUB_InitDone								:= FALSE;

				g_uControl_X_Axis.bEnableDrive				:= FALSE;
				g_uControl_X_Axis.bPosABSPosition			:= FALSE;
				//g_uControl_X_Axis.bStartManualMode		:= FALSE;

				g_uControl_Y_Axis.bEnableDrive				:= FALSE;
				g_uControl_Y_Axis.bPosABSPosition			:= FALSE;
				//g_uControl_Y_Axis.bStartManualMode		:= FALSE;

				//g_uControl_Front_Axis.bEnableDrive		:= FALSE;
				//g_uControl_Front_Axis.bAutomatic			:= FALSE;

				//g_uControl_Rear_Axis.bEnableDrive			:= FALSE;
				//g_uControl_Rear_Axis.bAutomatic			:= FALSE;

				g_uControl_Z_Axis.bEnableDrive				:= FALSE;
				//g_uControl_Z_Axis.bStartManualMode		:= FALSE;
				g_uControl_Z_Axis.bStartHoming				:= FALSE;
				g_uControl_Z_Axis.bPosABSPosition			:= FALSE;	(* Used only after axis has first been homed to its sensor *)

				g_uControl_R_Axis.bEnableDrive				:= FALSE;
				g_uControl_R_Axis.bPosABSPosition			:= FALSE;
				//g_uControl_R_Axis.bStartManualMode		:= FALSE;

				g_sMACH.sCleaningContainerControl.bPosExecute := FALSE;

		END_IF

		(* Continuous actions *)

		(* Transitions *)
		IF		g_bSUB_InitStart
		THEN
				g_sMACH.SUBInit.nStepCounter			:= C_INITIAL;
		END_IF

	(* --------------------------------------------------------------------------
	 * S000 C_INITIAL
	 *		OnEntry: Ready := FALSE
	 *		OnEntry: Busy  := TRUE
	 * T001 Always
	 * -------------------------------------------------------------------------- *)
	C_INITIAL:

		(* On Entry *)
		IF			bPulseStepCounter
		THEN
					g_sMACH.SUBInit.rWatchdogTime			:= 10 * 1000;
					g_sMACH.SUBInit.bSUBReady				:= FALSE;
					g_sMACH.SUBInit.bSUBBusy				:= TRUE;

					tDelayStep5.IN := FALSE;

					g_uControl_X_Axis.bEnableDrive		:= TRUE;
					g_uControl_Y_Axis.bEnableDrive		:= TRUE;
					g_uControl_Front_Axis.bEnableDrive	:= TRUE;
					g_uControl_Rear_Axis.bEnableDrive	:= TRUE;
					g_uControl_Z_Axis.bEnableDrive		:= TRUE;
					g_uControl_R_Axis.bEnableDrive		:= TRUE;

		END_IF

		(* Continuous actions *)
		Calc_BottomPos();	// Calculate Z bottom pos and pos above product

		IF g_sMACH.SUBInit.bAlmError THEN
			IF 	NOT g_uStatus_X_Axis.bDriveEnabled
				OR NOT g_uStatus_Y_Axis.bDriveEnabled
				OR NOT g_uStatus_Front_Axis.bDriveEnabled
				OR NOT g_uStatus_Rear_Axis.bDriveEnabled
			THEN
				g_sMACH.ERR.bXYNotEnabled := TRUE;
			END_IF
			IF NOT g_uStatus_Z_Axis.bDriveEnabled THEN
				g_sMACH.ERR.bZNotEnabled := TRUE;
			END_IF
			IF NOT g_uStatus_R_Axis.bDriveEnabled THEN
				g_sMACH.ERR.bRNotEnabled := TRUE;
			END_IF
		END_IF

		(* Transitions *)
		IF		g_uStatus_X_Axis.bDriveEnabled
			AND	g_uStatus_Y_Axis.bDriveEnabled
			AND	g_uStatus_Front_Axis.bDriveEnabled //bAutomaticEnabled
			AND	g_uStatus_Rear_Axis.bDriveEnabled //bAutomaticEnabled
			AND	g_uStatus_Z_Axis.bDriveEnabled
			AND	g_uStatus_R_Axis.bDriveEnabled
		THEN
					tDelayStep5.IN := TRUE;
					IF tDelayStep5.Q THEN
						tDelayStep5.IN := FALSE;
						g_sMACH.SUBInit.nStepCounter			:= 005;
					END_IF
		END_IF

	(* --------------------------------------------------------------------------
	 * S005 Start homing Z
	 * T010 Z axis busy
	 * -------------------------------------------------------------------------- *)
	005:

		(* On Entry *)
		IF		 bPulseStepCounter
		THEN
				g_sMACH.SUBInit.rWatchdogTime			:= 0;
				g_sMACH.SUBInit.rStepTime				:= 0;
				IF g_uStatus_Z_Axis.bHomePositionAvailable THEN
					g_uControl_Z_Axis.lrPosition			:= 0;
					g_uControl_Z_Axis.bPosABSPosition	:= TRUE;
				ELSE
					g_uControl_Z_Axis.bStartHoming	:= TRUE;
				END_IF
		END_IF

		(* Continuous actions *)

		(* Transitions *)
		IF			g_uStatus_Z_Axis.bHomingBusy
				OR	g_uStatus_Z_Axis.bMoveAbsDone
		THEN
					g_sMACH.SUBInit.nStepCounter				:= 010;
		END_IF

	(* --------------------------------------------------------------------------
	 * S010 Wait Z homing done
	 * T015 Z axis Homing done
	 * -------------------------------------------------------------------------- *)
	010:

		(* On Entry *)
		IF		 bPulseStepCounter
		THEN
				g_sMACH.SUBInit.rWatchdogTime		:= 0;
				g_sMACH.SUBInit.rStepTime				:= 0;
		END_IF

		(* Continuous actions *)

		(* Transitions *)
		IF			(g_uStatus_Z_Axis.bHomingDone OR g_uStatus_Z_Axis.bMoveAbsDone)
		THEN
					g_uControl_Z_Axis.bStartHoming		:= FALSE;
					g_uControl_Z_Axis.bPosABSPosition	:= FALSE;
					g_sMACH.SUBInit.nStepCounter			:= 015;
		END_IF

	(* --------------------------------------------------------------------------
	 * S015 Start homing R and cleaning cylinder down
	 * T020 R axis busy
	 * -------------------------------------------------------------------------- *)
	015:

		(* On Entry *)
		IF		 bPulseStepCounter
		THEN
				g_sMACH.SUBInit.rWatchdogTime		:= 0;
				g_sMACH.SUBInit.rStepTime			:= 500;
				g_uControl_R_Axis.lrPosition		:= 0;
				g_uControl_R_Axis.bPosABSPosition	:= TRUE;
				g_sMACH.sCleaningContainerControl.rTargetPosition := 0;
				g_sMACH.sCleaningContainerControl.bPosExecute := gMachConfig.bCleaningUnit;
		END_IF

		(* Continuous actions *)

		(* Transitions *)
		IF	NOT bWait
		THEN
					g_sMACH.SUBInit.nStepCounter				:= 020;
		END_IF

	(* --------------------------------------------------------------------------
	 * S020 Wait for R homing done
	 * T025 R-axis homing done
	 * -------------------------------------------------------------------------- *)
	020:

		(* On Entry *)
		IF		 bPulseStepCounter
		THEN
				g_sMACH.SUBInit.rWatchdogTime		:= 0;
				g_sMACH.SUBInit.rStepTime			:= 0;
		END_IF

		(* Continuous actions *)

		(* Transitions *)
		IF		g_uStatus_R_Axis.bMoveAbsDone
			AND (g_sMACH.sCleaningContainerStatus.rActualPosition = 0 OR NOT gMachConfig.bCleaningUnit)
		THEN
				g_uControl_R_Axis.bPosABSPosition	:= FALSE;
				g_sMACH.sCleaningContainerControl.bPosExecute	:= FALSE;
				g_sMACH.SUBInit.nStepCounter			:= 025;
		END_IF

	(* --------------------------------------------------------------------------
	 * S025 Start positioning Y to pre infeed position
	 * T030 Y axis ready
	 * -------------------------------------------------------------------------- *)
	025:

		(* On Entry *)
		IF		 bPulseStepCounter
		THEN
				g_sMACH.SUBInit.rWatchdogTime		:= 0;
				g_sMACH.SUBInit.rStepTime			:= 0;
				g_uControl_Y_Axis.lrPosition		:= I_rY_InfeedPrePosition;
				g_uControl_Y_Axis.bPosABSPosition	:= TRUE;
		END_IF

		(* Continuous actions *)

		(* Transitions *)
		IF			g_uStatus_Y_Axis.bMoveAbsDone
		THEN
					g_uControl_Y_Axis.bPosABSPosition	:= FALSE;
					g_sMACH.SUBInit.nStepCounter		:= 030;
		END_IF

	(* --------------------------------------------------------------------------
	 * S030 Start homing X
	 * T035 X axis ready
	 * -------------------------------------------------------------------------- *)
	030:

		(* On Entry *)
		IF		 bPulseStepCounter
		THEN
				g_sMACH.SUBInit.rWatchdogTime		:= 0;
				g_sMACH.SUBInit.rStepTime				:= 0;
				g_uControl_X_Axis.lrPosition			:= I_rX_InfeedPosition;
				g_uControl_X_Axis.bPosABSPosition	:= TRUE;
		END_IF

		(* Continuous actions *)

		(* Transitions *)
		IF			g_uStatus_X_Axis.bMoveAbsDone
		THEN
					g_uControl_X_Axis.bPosABSPosition	:= FALSE;
					g_sMACH.SUBInit.nStepCounter			:= 035;
		END_IF

	(* --------------------------------------------------------------------------
	 * S035 Start homing Y
	 * T040 Y axis ready
	 * -------------------------------------------------------------------------- *)
	035:

		(* On Entry *)
		IF		 bPulseStepCounter
		THEN
				g_sMACH.SUBInit.rWatchdogTime		:= 0;
				g_sMACH.SUBInit.rStepTime			:= 0;
				g_uControl_Y_Axis.lrPosition		:= I_rY_InfeedPosition;
				g_uControl_Y_Axis.bPosABSPosition	:= TRUE;
		END_IF

		(* Continuous actions *)

		(* Transitions *)
		IF			g_uStatus_Y_Axis.bMoveAbsDone
		THEN
					g_uControl_Y_Axis.bPosABSPosition	:= FALSE;
					g_sMACH.SUBInit.nStepCounter			:= 040;
		END_IF

	(* --------------------------------------------------------------------------
	 * S040 Stop manual mode of drives
	 * C_READY All axis out of manual mode
	 * -------------------------------------------------------------------------- *)
	040:

		(* On Entry *)
		IF		bPulseStepCounter
		THEN
				g_sMACH.SUBInit.rWatchdogTime		:= 0;
				g_sMACH.SUBInit.rStepTime				:= 400;
		END_IF

		(* Continuous actions *)
		IF NOT	bWait
		THEN
				(*g_uControl_X_Axis.bStartManualMode		:= FALSE;
				g_uControl_Y_Axis.bStartManualMode		:= FALSE;
				g_uControl_Front_Axis.bAutomatic			:= FALSE;
				g_uControl_Rear_Axis.bAutomatic			:= FALSE;
				g_uControl_Z_Axis.bStartManualMode		:= FALSE;
				g_uControl_R_Axis.bStartManualMode		:= FALSE;*)
		END_IF

		(* Transitions *)
		IF			g_uStatus_X_Axis.eStateAxis = L_MC1P_AXIS_STATE.StandStill
			AND 	g_uStatus_Y_Axis.eStateAxis = L_MC1P_AXIS_STATE.StandStill
			(*AND 	g_uStatus_Front_Axis.eStateAxis = L_MC1P_AXIS_STATE.StandStill
			AND 	g_uStatus_Rear_Axis.eStateAxis = L_MC1P_AXIS_STATE.StandStill*)
			AND 	g_uStatus_Z_Axis.eStateAxis = L_MC1P_AXIS_STATE.StandStill
			AND 	g_uStatus_R_Axis.eStateAxis = L_MC1P_AXIS_STATE.StandStill
		THEN
					g_uControl_X_Axis.bEnableDrive		:= FALSE;
					g_uControl_Y_Axis.bEnableDrive		:= FALSE;
					//g_uControl_Front_Axis.bEnableDrive	:= FALSE;
					//g_uControl_Rear_Axis.bEnableDrive	:= FALSE;
					g_uControl_Z_Axis.bEnableDrive		:= FALSE;
					g_uControl_R_Axis.bEnableDrive		:= FALSE;

					g_sMACH.SUBInit.nStepCounter				:= C_READY;
		END_IF

	(* --------------------------------------------------------------------------
	 * S998 C_READY
	 *		OnEntry: Ready		:= TRUE
	 *		OnEntry: Busy		 := FALSE
	 *		Always : Activate errorhandler
	 * T000 Never
	 * -------------------------------------------------------------------------- *)
	C_READY:

		(* On Entry *)
		IF			bPulseStepCounter
		THEN
					g_sMACH.SUBInit.rWatchdogTime	:= 0;
					g_sMACH.SUBInit.bSUBReady		:= TRUE;
					g_sMACH.SUBInit.bSUBBusy		:= FALSE;
		END_IF

		(* Continuous actions *)
		g_bSUB_InitDone		:= TRUE;

		(* Transitions *)
		IF			FALSE
		THEN
					g_sMACH.SUBInit.nStepCounter				:= C_INITIAL;
		END_IF

(* --------------------------------------------------------------------------
 * Illegal state
 * -------------------------------------------------------------------------- *)
ELSE
	(* Programming error: Illegal state *)
	g_sMACH.SUBInit.rWatchdogTime := 10;
END_CASE;

IF			g_sMACH.SUBInit.nStepCounter <> C_NOT_ACTIVE
THEN
	(* -------------------------------------------------------------------------
	 * Poststep Code
	 * ------------------------------------------------------------------------- *)
	;
END_IF

END_PROGRAM

(* ---- OutputControl.pou ---- *)
PROGRAM OutputControl
VAR
	tofResetSafety	: TOF;
END_VAR
%LANGUAGE ST
                        g_bDQ_LampStart				:= 		g_sMACH.ERR.bPressStartForManual
								OR	g_sMACH.ERR.bPressStartToCleanInit
								OR	(g_sMACH.ERR.bPressStartToCut AND NOT g_HMI_MachCommand.bScanMode)
								OR	g_sMACH.ERR.bPressStartToInit;
								//OR	g_bDI_MachineInSafePosition;

//Reset signal to safety
tofResetSafety(
	IN:=g_HMI_MachCommand.CMD.bResetEmergencyStop,
	PT:=T#250MS,
	Q=>g_bDQ_ResetSafety
);

g_HMI_MachCommand.CMD.bResetEmergencyStop := FALSE;	//Auto RESET-bit from HMI

//Start signal to safety
g_bDQ_LightCurtainActive := InputControl.bStartPressed;

(*thirth module *)
g_byOutputs_Module_00.0		:= g_bDQ_ResetSafety;
g_byOutputs_Module_00.1		:= g_bDQ_LightCurtainActive;
g_byOutputs_Module_00.2		:= g_bDQ_MainValve;
g_byOutputs_Module_00.3		:= g_bDQ_Ultrasonic1;
g_byOutputs_Module_00.4		:= g_bDQ_LampStart;
g_byOutputs_Module_00.5		:= g_bDQ_Servo_Power_Reset;
g_byOutputs_Module_00.6		:= g_bDQ_Buzzer;
g_byOutputs_Module_00.7		:= g_bDQ_Spare_17;

(*fourth module *)
g_byOutputs_Module_01.0		:= g_bDQ_CleaningContainerUp;
g_byOutputs_Module_01.1		:= g_bDQ_CleaningContainerDown;
g_byOutputs_Module_01.2		:= g_bDQ_CleaningAirValve;
g_byOutputs_Module_01.3		:= g_bDQ_CleaningWaterValve;
g_byOutputs_Module_01.4		:= g_bDQ_Spare_24;
g_byOutputs_Module_01.5		:= g_bDQ_Spare_25;
g_byOutputs_Module_01.6		:= g_bDQ_Spare_26;
g_byOutputs_Module_01.7		:= g_bDQ_Spare_27;

(*sixth module *)
g_wOutputs_Module_00		:= TO_WORD((TO_REAL(g_iAQ_UltrasonicPower)/100)*16384);
g_wOutputs_Module_01		:= TO_WORD((TO_REAL(g_iAQ_Spare_01)/100)*16384);

(*Data to IO *)
//Digital
%QB1						:= g_byOutputs_Module_00;
%QB2						:= g_byOutputs_Module_01;
//Analog
%QW2						:= g_wOutputs_Module_00;
%QW3						:= g_wOutputs_Module_01;

END_PROGRAM
